(* PLC project multi-phase-flow-facility, Generated TextualNotationConverter 1.0 *)
(* stored: creationDateTime 2025-07-30T12:00:00, modificationDateTime 2025-01-30T12:00:00 *)

FUNCTION_BLOCK ANALOG_IN
  VAR_INPUT
    Name : STRING;
    Description : STRING;
    Raw_Signal : REAL;
    PV_High : REAL;
    PV_Low : REAL;
    Scaling_Slope : REAL;
    Scaling_Offset : REAL;
    Alarm_Enable : BOOL;
  END_VAR
  VAR_OUTPUT
    PV : REAL;
    High_Alarm : BOOL;
    Low_Alarm : BOOL;
    General_Fault : BOOL;
  END_VAR

            
          
END_FUNCTION_BLOCK

FUNCTION_BLOCK PID_BASIC
  VAR_INPUT
    Name : STRING;
    Description : STRING;
    AUTO : BOOL;
    PV : REAL;
    SP : REAL;
    MV_MIN : REAL;
    MV_MAX : REAL;
    X0 : REAL;
    KP : REAL;
    TR : REAL;
    TD : REAL;
    PV_High : REAL;
    PV_Low : REAL;
    Deviation_Limit : REAL;
    Inhibit : BOOL;
  END_VAR
  VAR_OUTPUT
    PV_High_Alarm : BOOL;
    PV_Low_Alarm : BOOL;
    Deviation_Alarm : BOOL;
    XOUT : REAL;
  END_VAR

            
          
END_FUNCTION_BLOCK

FUNCTION_BLOCK RATIO_CONTROL
  VAR_INPUT
    Name : STRING;
    Description : STRING;
    Auto : BOOL;
    PrimaryPV : REAL;
    SecondaryPV : REAL;
    RatioSP : REAL;
    Bias : REAL;
    TrimKp : REAL;
    TrimTi : STRING;
    MV_MIN : REAL;
    MV_MAX : REAL;
    ManOut : REAL;
    Inhibit : BOOL;
  END_VAR
  VAR_OUTPUT
    SlaveSP : REAL;
    ActiveRatio : REAL;
    RatioErr : REAL;
  END_VAR

            
          
END_FUNCTION_BLOCK

FUNCTION_BLOCK VALVE_ELECTRIC
  VAR_INPUT
    Name : STRING;
    Description : STRING;
    Control_Signal : REAL;
    Manual_Mode : BOOL;
    Manual_Position : REAL;
    Open_Limit : REAL;
    Close_Limit : REAL;
    Timeout : STRING;
    Inhibit : BOOL;
  END_VAR
  VAR_OUTPUT
    Valve_Position : REAL;
    Feedback_Pos : REAL;
    Valve_Moving : BOOL;
    Position_Error : BOOL;
    Alarm : BOOL;
  END_VAR

            
          
END_FUNCTION_BLOCK

PROGRAM Section2
  VAR
    FT404_GasFlow_PV : REAL;
    FT406_LiqFlow_PV : REAL;
    PT403_SepPressure_PV : REAL;
    PT408_AuxPressure_PV : REAL;
    FIC406_LiqFlow_SP_From_FFIC402 : REAL;
  END_VAR
  VAR
    FT-404 : ANALOG_IN;
    FT-406 : ANALOG_IN;
    PT-403 : ANALOG_IN;
    PT-408 : ANALOG_IN;
    FFIC-402 : RATIO_CONTROL;
    FIC-406 : PID_BASIC;
    PIC-401 : PID_BASIC;
    CV-406 : VALVE_ELECTRIC;
    CV-401 : VALVE_ELECTRIC;
  END_VAR

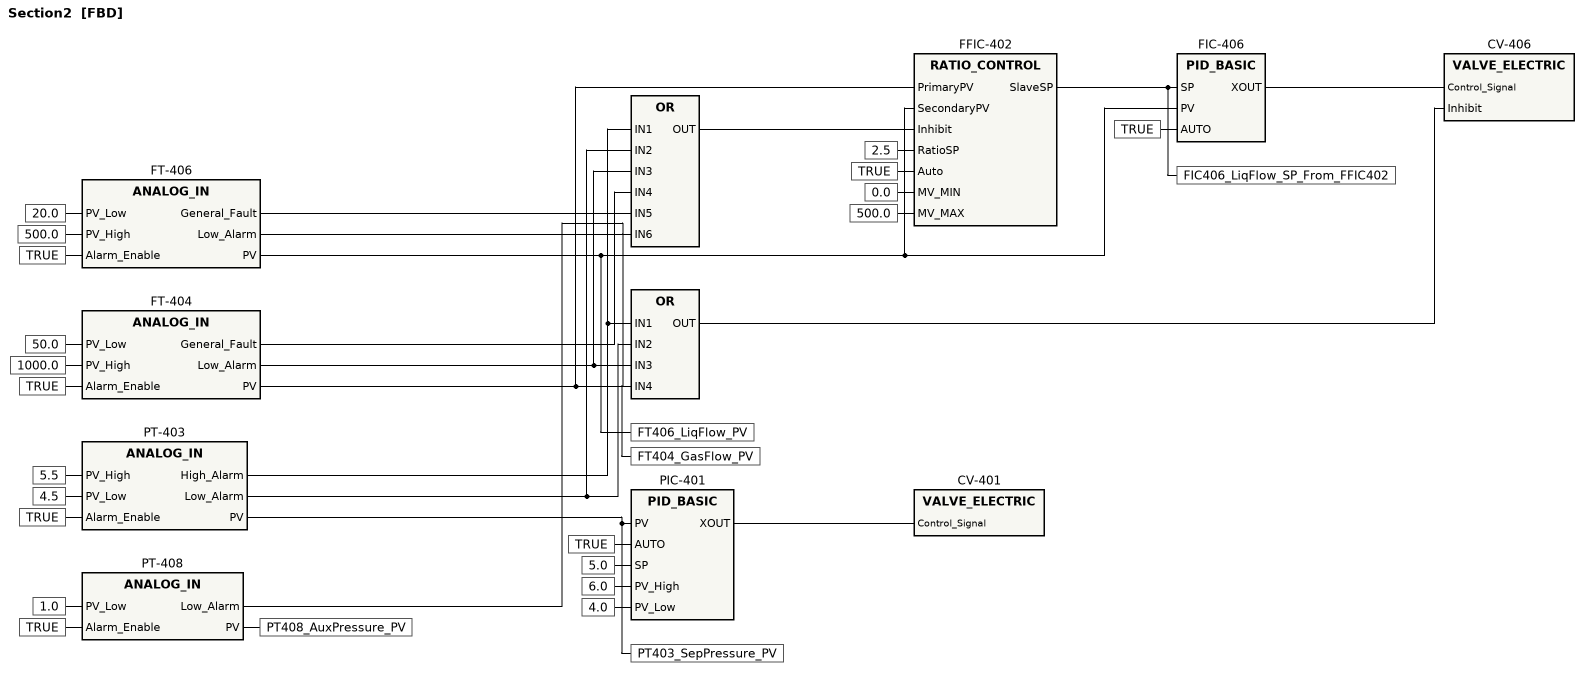
(* FBD diagram, written out as Structured Text *)
FT-404(PV_Low := 50.0, PV_High := 1000.0, Alarm_Enable := TRUE);
FT-406(PV_Low := 20.0, PV_High := 500.0, Alarm_Enable := TRUE);
PT-403(PV_High := 5.5, PV_Low := 4.5, Alarm_Enable := TRUE);
PT-408(PV_Low := 1.0, Alarm_Enable := TRUE);
FFIC-402(PrimaryPV := FT-404.PV, SecondaryPV := FT-406.PV, Inhibit := PT-403.High_Alarm OR PT-403.Low_Alarm OR FT-404.Low_Alarm OR FT-404.General_Fault OR FT-406.General_Fault OR PT-408.Low_Alarm, RatioSP := 2.5, Auto := TRUE, MV_MIN := 0.0, MV_MAX := 500.0);
FIC406_LiqFlow_SP_From_FFIC402 := FFIC-402.SlaveSP;
FT404_GasFlow_PV := FT-404.PV;
FT406_LiqFlow_PV := FT-406.PV;
PT403_SepPressure_PV := PT-403.PV;
PT408_AuxPressure_PV := PT-408.PV;
FIC-406(SP := FFIC-402.SlaveSP, PV := FT-406.PV, AUTO := TRUE);
PIC-401(PV := PT-403.PV, AUTO := TRUE, SP := 5.0, PV_High := 6.0, PV_Low := 4.0);
CV-406(Control_Signal := FIC-406.XOUT, Inhibit := PT-403.High_Alarm OR PT-403.Low_Alarm OR FT-404.Low_Alarm OR FT-406.Low_Alarm);
CV-401(Control_Signal := PIC-401.XOUT);
END_PROGRAM

FUNCTION_BLOCK BOOL_IN
  VAR_INPUT
    Name : STRING;
    Description : STRING;
    Bool_In : BOOL;
    Alarm_OnTrue : BOOL;
    Alarm_OnFalse : BOOL;
    Latch_Enable : BOOL;
    Reset_Latch : BOOL;
  END_VAR
  VAR_OUTPUT
    Bool_Out : BOOL;
    Alarm_Active : BOOL;
    Latched_Status : BOOL;
  END_VAR

            
          
END_FUNCTION_BLOCK

FUNCTION_BLOCK DIGITAL_IN
  VAR_INPUT
    Name : STRING;
    Description : STRING;
    DI_Raw : BOOL;
    DebounceTime : STRING;
    EnableAlarm : BOOL;
  END_VAR
  VAR_OUTPUT
    DI_Out : BOOL;
    Fault_State : BOOL;
  END_VAR

            
          
END_FUNCTION_BLOCK

FUNCTION_BLOCK DUTY_STANDBY
  VAR_INPUT
    Name : STRING;
    Description : STRING;
    Enable : BOOL;
    StartRequest : BOOL;
    AlternateEnable : BOOL;
    ForcePumpA : BOOL;
    ForcePumpB : BOOL;
    DutyElapsed : BOOL;
    MinRunElapsed : BOOL;
    SwitchoverDelayElapsed : BOOL;
    StartTimeoutElapsed : BOOL;
    PumpA_RunFB : BOOL;
    PumpB_RunFB : BOOL;
    PumpA_Fault : BOOL;
    PumpB_Fault : BOOL;
    Reset : BOOL;
    Inhibit : BOOL;
  END_VAR
  VAR_OUTPUT
    CmdPumpA : BOOL;
    CmdPumpB : BOOL;
    ActiveIsA : BOOL;
    SwitchedDueToDuty : BOOL;
    SwitchedDueToFailure : BOOL;
    Alarm_FailedStart_A : BOOL;
    Alarm_FailedStart_B : BOOL;
    Alarm_NoAvailablePump : BOOL;
  END_VAR

            
          
END_FUNCTION_BLOCK

FUNCTION_BLOCK MOTOR_2SPD
  VAR_INPUT
    Name : STRING;
    Description : STRING;
    Start_Cmd : BOOL;
    Stop_Cmd : BOOL;
    Speed_High_Cmd : BOOL;
    Speed_Low_Cmd : BOOL;
    Inhibit : BOOL;
  END_VAR
  VAR_OUTPUT
    Motor_Start_Out : BOOL;
    FB_Running : BOOL;
    FB_Trip : BOOL;
    FB_HighSpeed : BOOL;
    FB_LowSpeed : BOOL;
    Alarm_Speed_Error : BOOL;
  END_VAR

            
          
END_FUNCTION_BLOCK

FUNCTION_BLOCK MOTOR_ON_OFF
  VAR_INPUT
    Name : STRING;
    Description : STRING;
    Start_Cmd : BOOL;
    Stop_Cmd : BOOL;
    Start_Delay : STRING;
    MinRunTime : STRING;
    Inhibit : BOOL;
  END_VAR
  VAR_OUTPUT
    Motor_Start_Out : BOOL;
    FB_Running : BOOL;
    FB_Trip : BOOL;
    Alarm_Start_Fail : BOOL;
    Alarm_Stop_Fail : BOOL;
  END_VAR

            
          
END_FUNCTION_BLOCK

FUNCTION_BLOCK MOTOR_VSD
  VAR_INPUT
    Name : STRING;
    Description : STRING;
    Start_Cmd : BOOL;
    Stop_Cmd : BOOL;
    Speed_SP : REAL;
    Accel_Ramp : STRING;
    Decel_Ramp : STRING;
    Inhibit : BOOL;
  END_VAR
  VAR_OUTPUT
    Speed_Out : REAL;
    FB_Running : BOOL;
    FB_Fault : BOOL;
    FB_Ready : BOOL;
    FB_ActualSpeed : REAL;
    Alarm_Speed_Deviation : BOOL;
    Alarm_Comm_Fail : BOOL;
  END_VAR

            
          
END_FUNCTION_BLOCK

FUNCTION_BLOCK SPLIT_RANGE
  VAR_INPUT
    Name : STRING;
    Description : STRING;
    IN : REAL;
    Split_Point : REAL;
    Output1_Start : REAL;
    Output1_End : REAL;
    Output2_Start : REAL;
    Output2_End : REAL;
  END_VAR
  VAR_OUTPUT
    OUT1 : REAL;
    OUT2 : REAL;
  END_VAR

            
          
END_FUNCTION_BLOCK

FUNCTION_BLOCK VALVE_ON_OFF
  VAR_INPUT
    Name : STRING;
    Description : STRING;
    Open_Cmd : BOOL;
    Close_Cmd : BOOL;
    Timeout : STRING;
    Inhibit : BOOL;
  END_VAR
  VAR_OUTPUT
    FB_Opened : BOOL;
    FB_Closed : BOOL;
    Valve_Open_Out : BOOL;
    Valve_Close_Out : BOOL;
    Alarm_Position_Error : BOOL;
    Alarm_General : BOOL;
  END_VAR

            
          
END_FUNCTION_BLOCK

FUNCTION_BLOCK VOTING_ANALOG
  VAR_INPUT
    Name : STRING;
    Description : STRING;
    Input1 : REAL;
    Input2 : REAL;
    Input3 : REAL;
    Deviation_Limit : REAL;
    Voting_Scheme : STRING;
    EnableAlarm : BOOL;
    Inhibit : BOOL;
  END_VAR
  VAR_OUTPUT
    Voted_Output : REAL;
    Sensor1_Fault : BOOL;
    Sensor2_Fault : BOOL;
    Sensor3_Fault : BOOL;
    Alarm_Voting_Error : BOOL;
    Healthy_Sensors_Count : INT;
  END_VAR

            
          
END_FUNCTION_BLOCK

PROGRAM Section3
  VAR
    PT501_Pressure_PV : REAL;
    LI502_Level_PV : REAL;
    PIC501_Output_To_FV102 : REAL;
  END_VAR
  VAR
    PT-501 : ANALOG_IN;
    LI-502 : ANALOG_IN;
    PIC-501 : PID_BASIC;
    FV-102 : VALVE_ELECTRIC;
  END_VAR
  VAR  (* added by the conversion: wires and edge detectors of the diagram *)
    _OR37_OUT : BOOL;
  END_VAR

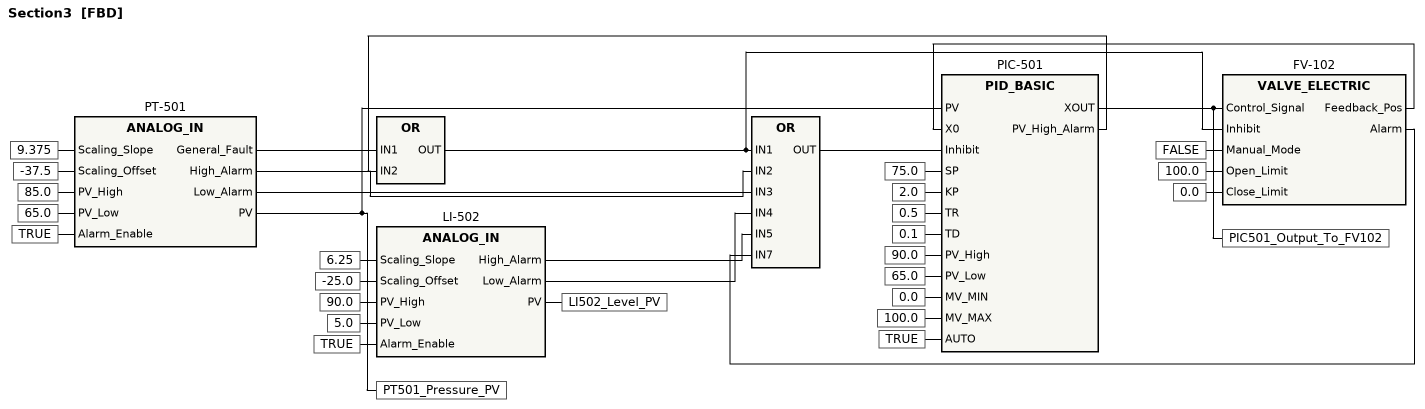
(* FBD diagram, written out as Structured Text *)
LI-502(Scaling_Slope := 6.25, Scaling_Offset := -25.0, PV_High := 90.0, PV_Low := 5.0, Alarm_Enable := TRUE);
LI502_Level_PV := LI-502.PV;
PT-501(Scaling_Slope := 9.375, Scaling_Offset := -37.5, PV_High := 85.0, PV_Low := 65.0, Alarm_Enable := TRUE);
_OR37_OUT := PT-501.General_Fault OR PIC-501.PV_High_Alarm;
FV-102(Control_Signal := PIC-501.XOUT, Inhibit := _OR37_OUT, Manual_Mode := FALSE, Open_Limit := 100.0, Close_Limit := 0.0);
PIC-501(PV := PT-501.PV, X0 := FV-102.Feedback_Pos, Inhibit := _OR37_OUT OR PT-501.High_Alarm OR PT-501.Low_Alarm OR LI-502.Low_Alarm OR LI-502.High_Alarm OR FV-102.Alarm, SP := 75.0, KP := 2.0, TR := 0.5, TD := 0.1, PV_High := 90.0, PV_Low := 65.0, MV_MIN := 0.0, MV_MAX := 100.0, AUTO := TRUE);
PIC501_Output_To_FV102 := PIC-501.XOUT;
PT501_Pressure_PV := PT-501.PV;
END_PROGRAM

PROGRAM Section4
  VAR
    LI201_Raw_mA : REAL;
    XV010_OpenSw_Raw : BOOL;
    XV011_OpenSw_Raw : BOOL;
    LI201_Level_PV_Pct : REAL;
    FIC302_MV_To_FV101_Pct : REAL;
    FV101_Feedback_Position_Pct : REAL;
  END_VAR
  VAR
    FIC-302 : PID_BASIC;
    FV-101 : VALVE_ELECTRIC;
    LI-201 : ANALOG_IN;
    XV-010-OPEN_FB : DIGITAL_IN;
    XV-011-OPEN_FB : DIGITAL_IN;
  END_VAR
  VAR  (* added by the conversion: wires and edge detectors of the diagram *)
    _AND68_OUT : BOOL;
  END_VAR

(* FBD diagram, written out as Structured Text *)
LI-201(Raw_Signal := LI201_Raw_mA, Alarm_Enable := TRUE, PV_High := 80.0, PV_Low := 20.0, Scaling_Slope := 6.25, Scaling_Offset := -25.0);
XV-010-OPEN_FB(DI_Raw := XV010_OpenSw_Raw);
XV-011-OPEN_FB(DI_Raw := XV011_OpenSw_Raw);
_AND68_OUT := XV-010-OPEN_FB.DI_Out AND XV-011-OPEN_FB.DI_Out;
FIC-302(PV := LI-201.PV, AUTO := NOT LI-201.General_Fault AND _AND68_OUT, SP := 70.0, MV_MIN := 0.0, MV_MAX := 100.0, X0 := 25.0, KP := 1.8, TR := 2.0, TD := 0.3, PV_High := 90.0, PV_Low := 20.0);
FIC302_MV_To_FV101_Pct := FIC-302.XOUT;
FV-101(Control_Signal := FIC-302.XOUT, Manual_Mode := NOT _AND68_OUT OR FIC-302.PV_High_Alarm, Open_Limit := 100.0, Close_Limit := 0.0, Manual_Position := 0.0);
FV101_Feedback_Position_Pct := FV-101.Feedback_Pos;
LI201_Level_PV_Pct := LI-201.PV;
END_PROGRAM

PROGRAM Section5
  VAR
    FIC101_MV_PCT : REAL;
    FIC102_MV_PCT : REAL;
    P001_Speed_AO_PCT : REAL;
    P001_Start_Cmd : BOOL;
    P001_Stop_Cmd : BOOL;
    FT102_FlowOK_Thresh : REAL;
    ValveOpenFB_Threshold : REAL;
    LevelOK_Threshold : REAL;
    FIC101_Deviation_Alarm_15s : BOOL;
    FIC102_Deviation_Alarm_15s : BOOL;
  END_VAR
  VAR
    FT-102 : ANALOG_IN;
    FT-104 : ANALOG_IN;
    LI-101 : ANALOG_IN;
    FIC-101 : PID_BASIC;
    FIC-102 : PID_BASIC;
    FV-103 : VALVE_ELECTRIC;
    P-001 : MOTOR_VSD;
    FlowOK_TON : TON;
    FIC101_Dev_TON : TON;
    FIC102_Dev_TON : TON;
  END_VAR

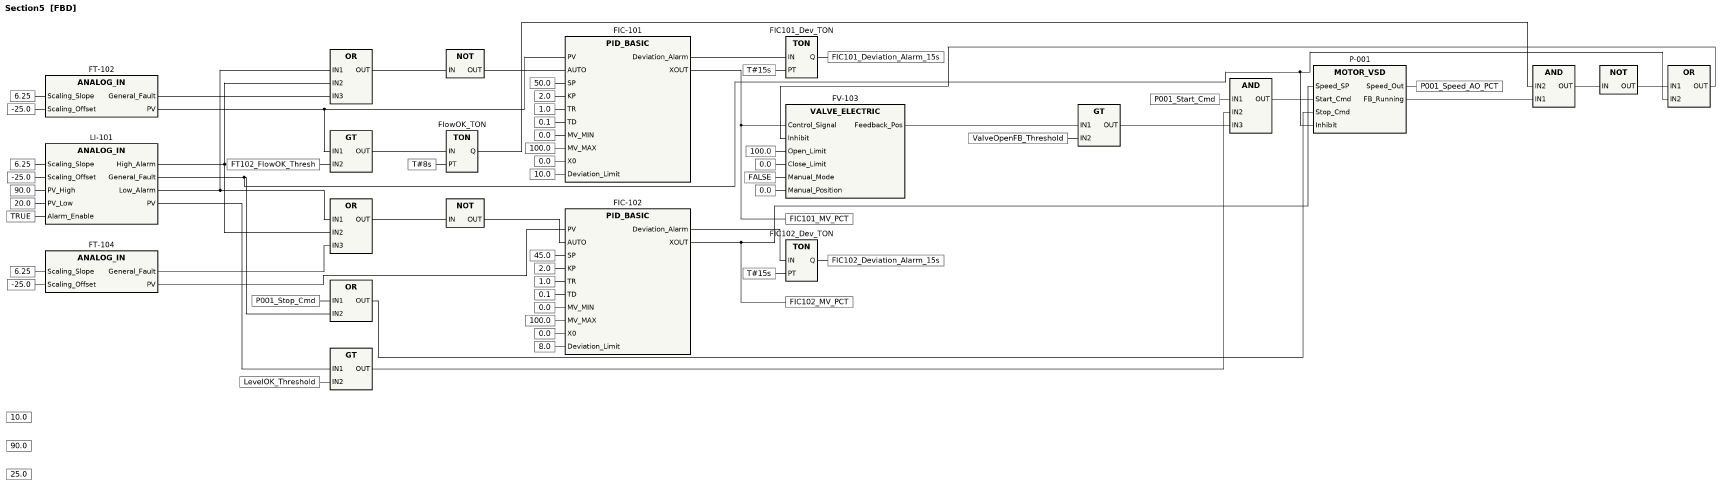
(* FBD diagram, written out as Structured Text *)
FT-102(Scaling_Slope := 6.25, Scaling_Offset := -25.0);
LI-101(Scaling_Slope := 6.25, Scaling_Offset := -25.0, PV_High := 90.0, PV_Low := 20.0, Alarm_Enable := TRUE);
FIC-101(PV := FT-102.PV, AUTO := NOT (LI-101.Low_Alarm OR LI-101.High_Alarm OR FT-102.General_Fault), SP := 50.0, KP := 2.0, TR := 1.0, TD := 0.1, MV_MIN := 0.0, MV_MAX := 100.0, X0 := 0.0, Deviation_Limit := 10.0);
FIC101_Dev_TON(IN := FIC-101.Deviation_Alarm, PT := T#15s);
FIC101_Deviation_Alarm_15s := FIC101_Dev_TON.Q;
FIC101_MV_PCT := FIC-101.XOUT;
FT-104(Scaling_Slope := 6.25, Scaling_Offset := -25.0);
FIC-102(PV := FT-104.PV, AUTO := NOT (LI-101.Low_Alarm OR LI-101.High_Alarm OR FT-104.General_Fault), SP := 45.0, KP := 2.0, TR := 1.0, TD := 0.1, MV_MIN := 0.0, MV_MAX := 100.0, X0 := 0.0, Deviation_Limit := 8.0);
FIC102_Dev_TON(IN := FIC-102.Deviation_Alarm, PT := T#15s);
FIC102_Deviation_Alarm_15s := FIC102_Dev_TON.Q;
FIC102_MV_PCT := FIC-102.XOUT;
FlowOK_TON(IN := FT-102.PV > FT102_FlowOK_Thresh, PT := T#8s);
FV-103(Control_Signal := FIC-101.XOUT, Inhibit := NOT (FlowOK_TON.Q AND P-001.FB_Running) OR LI-101.General_Fault, Open_Limit := 100.0, Close_Limit := 0.0, Manual_Mode := FALSE, Manual_Position := 0.0);
P-001(Speed_SP := FIC-102.XOUT, Start_Cmd := P001_Start_Cmd AND LI-101.PV > LevelOK_Threshold AND FV-103.Feedback_Pos > ValveOpenFB_Threshold, Stop_Cmd := P001_Stop_Cmd OR LI-101.General_Fault, Inhibit := LI-101.General_Fault);
P001_Speed_AO_PCT := P-001.Speed_Out;
(* drawn but not wired to any output: 10.0, 90.0, 25.0 *)
END_PROGRAM

PROGRAM Section6
  VAR
    FT105_FlowRate_gpm : REAL;
    LI503_Level_Pct : REAL;
    P001_Running_Permissive : BOOL;
  END_VAR
  VAR
    FT-105 : ANALOG_IN;
    LI-503 : ANALOG_IN;
    LIC-502 : PID_BASIC;
    LIC-503 : PID_BASIC;
    LVC-502 : VALVE_ELECTRIC;
    LVC-507 : VALVE_ELECTRIC;
    P-001 : MOTOR_ON_OFF;
  END_VAR
  VAR  (* added by the conversion: wires and edge detectors of the diagram *)
    _NOT168_OUT : BOOL;
    _OR169_OUT : BOOL;
    _OR170_OUT : BOOL;
  END_VAR

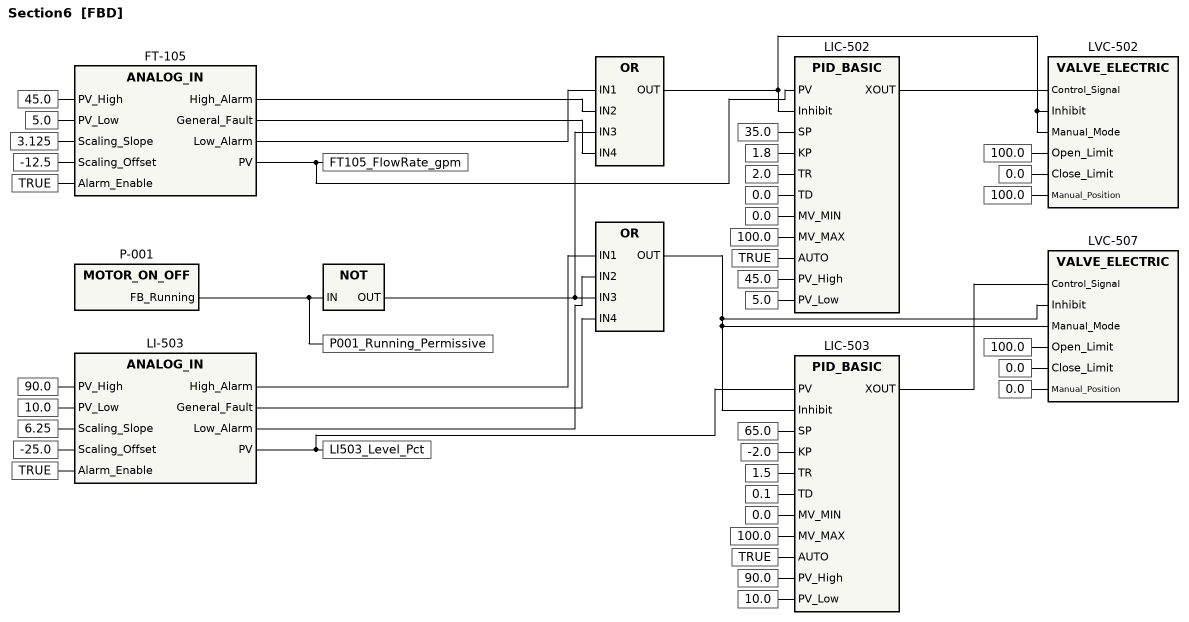
(* FBD diagram, written out as Structured Text *)
FT-105(PV_High := 45.0, PV_Low := 5.0, Scaling_Slope := 3.125, Scaling_Offset := -12.5, Alarm_Enable := TRUE);
FT105_FlowRate_gpm := FT-105.PV;
LI-503(PV_High := 90.0, PV_Low := 10.0, Scaling_Slope := 6.25, Scaling_Offset := -25.0, Alarm_Enable := TRUE);
LI503_Level_Pct := LI-503.PV;
P-001();
P001_Running_Permissive := P-001.FB_Running;
_NOT168_OUT := NOT P-001.FB_Running;
_OR169_OUT := LI-503.High_Alarm OR LI-503.Low_Alarm OR _NOT168_OUT OR LI-503.General_Fault;
_OR170_OUT := FT-105.Low_Alarm OR FT-105.High_Alarm OR _NOT168_OUT OR FT-105.General_Fault;
LIC-502(PV := FT-105.PV, Inhibit := _OR170_OUT, SP := 35.0, KP := 1.8, TR := 2.0, TD := 0.0, MV_MIN := 0.0, MV_MAX := 100.0, AUTO := TRUE, PV_High := 45.0, PV_Low := 5.0);
LIC-503(PV := LI-503.PV, Inhibit := _OR169_OUT, SP := 65.0, KP := -2.0, TR := 1.5, TD := 0.1, MV_MIN := 0.0, MV_MAX := 100.0, AUTO := TRUE, PV_High := 90.0, PV_Low := 10.0);
LVC-502(Control_Signal := LIC-502.XOUT, Inhibit := _OR170_OUT, Manual_Mode := _OR170_OUT, Open_Limit := 100.0, Close_Limit := 0.0, Manual_Position := 100.0);
LVC-507(Control_Signal := LIC-503.XOUT, Inhibit := _OR169_OUT, Manual_Mode := _OR169_OUT, Open_Limit := 100.0, Close_Limit := 0.0, Manual_Position := 0.0);
END_PROGRAM

PROGRAM Section7
  VAR
    PIT106_Raw_mA : REAL;
    CompressorRunPermissive : BOOL;
    PIT106_PressureBar : REAL;
    PIC105_MV_Percent : REAL;
  END_VAR
  VAR
    PIT-106 : ANALOG_IN;
    COMP-RUN-PERM : BOOL_IN;
    PIC-105 : PID_BASIC;
    V-010 : VALVE_ELECTRIC;
    CompStartupDelay : TON;
  END_VAR
  VAR  (* added by the conversion: wires and edge detectors of the diagram *)
    _OR216_OUT : BOOL;
  END_VAR

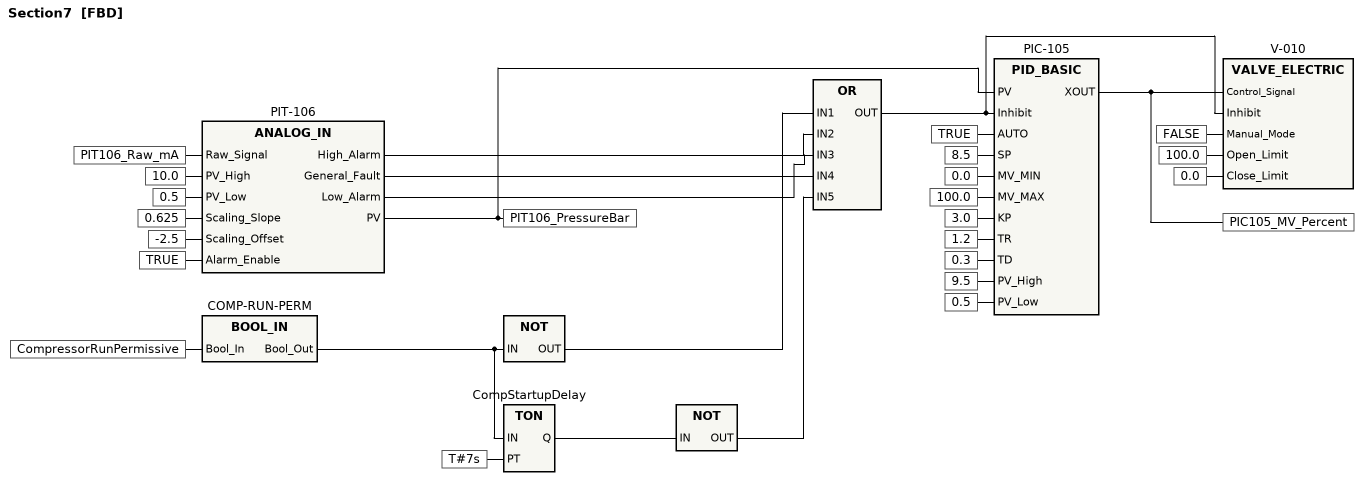
(* FBD diagram, written out as Structured Text *)
PIT-106(Raw_Signal := PIT106_Raw_mA, PV_High := 10.0, PV_Low := 0.5, Scaling_Slope := 0.625, Scaling_Offset := -2.5, Alarm_Enable := TRUE);
COMP-RUN-PERM(Bool_In := CompressorRunPermissive);
CompStartupDelay(IN := COMP-RUN-PERM.Bool_Out, PT := T#7s);
_OR216_OUT := NOT COMP-RUN-PERM.Bool_Out OR PIT-106.High_Alarm OR PIT-106.Low_Alarm OR PIT-106.General_Fault OR NOT CompStartupDelay.Q;
PIC-105(PV := PIT-106.PV, Inhibit := _OR216_OUT, AUTO := TRUE, SP := 8.5, MV_MIN := 0.0, MV_MAX := 100.0, KP := 3.0, TR := 1.2, TD := 0.3, PV_High := 9.5, PV_Low := 0.5);
PIC105_MV_Percent := PIC-105.XOUT;
PIT106_PressureBar := PIT-106.PV;
V-010(Control_Signal := PIC-105.XOUT, Inhibit := _OR216_OUT, Manual_Mode := FALSE, Open_Limit := 100.0, Close_Limit := 0.0);
END_PROGRAM

CONFIGURATION Config0
  RESOURCE Res0 ON PLC
    TASK task0(INTERVAL := T#20ms, PRIORITY := 0);
    PROGRAM instance0 WITH task0 : Section2;
    PROGRAM instance_1 WITH task0 : Section3;
    PROGRAM instance_2 WITH task0 : Section4;
    PROGRAM instance_3 WITH task0 : Section5;
    PROGRAM instance_4 WITH task0 : Section6;
    PROGRAM instance_5 WITH task0 : Section7;
  END_RESOURCE
END_CONFIGURATION
